// TwinCAT 3 PLC project PLC_wash
// ProgramVersion: 3.1.4022.3
// libraries:
//   Tc2_Standard, * (Beckhoff Automation GmbH)
//   Tc2_System, * (Beckhoff Automation GmbH)
//   Tc3_Module, * (Beckhoff Automation GmbH)
//   VisuSymbols,3.5.10.0,System
// project tree:
//   / GlobalTextList.TcGTLO, PlcTask.TcTTO (not stored), Visualization Manager.TcVMO (not stored)
//   GVLs/ GVL_IO.TcGVL
//   POUs/ MAIN.TcPOU
//   VISUs/ Visualization.TcVIS
// real-time tasks:
//   TASK PlcTask: cycle T#10ms, priority 20, ADS port 350

// ---- GVLs/GVL_IO.TcGVL
{attribute 'qualified_only'}
VAR_GLOBAL
	Fill_valve :BOOL;   // Fill water 
	Drain_valve:BOOL;   // Drain
	SpinMotor  :BOOL;   // Spin Motor
	AgitateMotor: BOOL; // Washing
	PumpOutMotor: BOOL; // Pump motor
    HeaterControl: BOOL; // Optional	
	StartWashing : BOOL;
END_VAR

// ---- POUs/MAIN.TcPOU
PROGRAM MAIN
VAR
	state_Fill:BOOL;
	State_Wash:BOOL;
	State_Rinse:BOOL;
	State_Spin:BOOL;
	Warmwash:BOOL;
	timertime:TIME := T#2000MS;
	Processtime:TON;
	start:BOOL;
	trigger:R_TRIG;
	
	step: INT;
END_VAR

// Your program  comes here ..... 
Processtime(IN:=start, PT:=timertime);
trigger(clk:=gvl_io.StartWashing);


//case: start true dan states true, dan
CASE step OF
	0:
	IF trigger.Q THEN
		start:=TRUE;
		state_Fill:=TRUE;
		gvl_IO.Fill_valve:=TRUE;	
	END_IF
	IF Processtime.Q THEN
		start:=FALSE;
		state_Fill:=FALSE;
		gvl_io.Fill_valve:= FALSE;
		step:=step+1;
	END_IF
	
	1:	
	IF Warmwash THEN
		timertime:=T#6000MS;
		start:=TRUE;
		State_Wash:=TRUE;
		gvl_io.AgitateMotor:=TRUE;
		gvl_io.HeaterControl:=TRUE;
	
	IF	Processtime.Q THEN
		start:=FALSE;
		gvl_io.AgitateMotor:=FALSE;
		gvl_io.HeaterControl:=FALSE;
		step:=step+1;
	END_IF	
		
	END_IF
	
	IF WarmWash=FALSE THEN
		start:=TRUE;
	State_Wash:=TRUE;
	gvl_io.AgitateMotor:=TRUE;
	
	IF	Processtime.Q THEN
		start:=FALSE;
		gvl_io.AgitateMotor:=FALSE;
		step:=step+1;
	END_IF		
	END_IF

	2:
	timertime:=T#2000ms;
	start:=TRUE;
	gvl_io.Drain_valve:=TRUE;
	gvl_io.PumpOutMotor:=TRUE;
	
		IF	Processtime.Q THEN
		start:=FALSE;
		State_Wash:=FALSE;
		gvl_io.Drain_valve:=FALSE;
		gvl_io.PumpOutMotor:=FALSE;
		step:=step+1;
	END_IF	
	
	3:
	start:=TRUE;
	State_Rinse:=TRUE;
	gvl_io.Fill_valve:=TRUE;
	
		IF	Processtime.Q THEN
		start:=FALSE;
		gvl_io.Fill_valve:=FALSE;
		step:=step+1;
	END_IF	
	
	4:
	start:=TRUE;
	gvl_io.AgitateMotor:=TRUE;
	
		IF	Processtime.Q THEN
		start:=FALSE;
		gvl_io.AgitateMotor:=FALSE;
		state_Rinse:=FALSE;
		step:=step+1;
	END_IF	
	5:
	start:=TRUE;
	State_Spin:=TRUE;
	gvl_io.Drain_valve := TRUE;
	gvl_io.SpinMotor:=TRUE;
	gvl_io.PumpOutMotor:=TRUE;
	
		IF	Processtime.Q THEN
		start:=FALSE;
		State_Spin:=FALSE;
		gvl_io.Drain_valve:=FALSE;
		gvl_io.SpinMotor:=FALSE;
		gvl_io.PumpOutMotor:=FALSE;
		step:=0;
	END_IF	
	
END_CASE

END_PROGRAM

// ---- GlobalTextList.TcGTLO
TEXTLIST GlobalTextList
  869 = '%s'
  746 = 'Agitate Motor'
  130 = 'Drain  Valve'
  802 = 'Fill'
  4 = 'Fill Valve'
  757 = 'Heater'
  21 = 'P'
  599 = 'Processtime.ET'
  355 = 'Pump Out Motor'
  679 = 'Rinse'
  546 = 'Spin'
  353 = 'Spin Motor'
  372 = 'Start/Stop'
  733 = 'Warm Washing'
  363 = 'Wash'
END_TEXTLIST

// ---- VISUs/Visualization.TcVIS
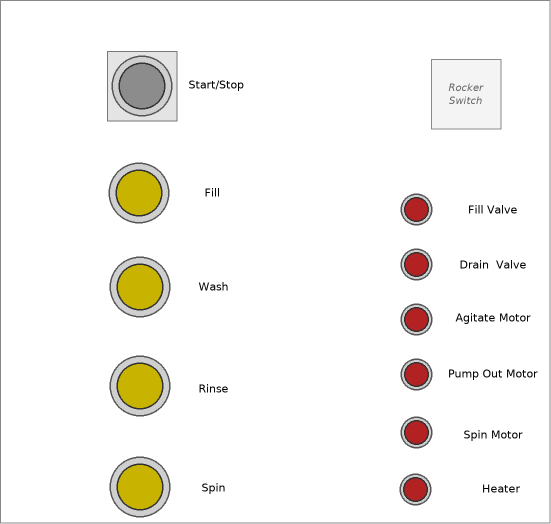
VISUALIZATION Visualization  // 551x524
    Lamp1 (104,158 70x70), variable: MAIN.state_Fill, style: Lamp-Lamp1-Yellow
    Lamp1 (105,252 70x70), variable: MAIN.State_Wash, style: Lamp-Lamp1-Yellow
    Lamp1 (105,351 70x70), variable: MAIN.State_Rinse, style: Lamp-Lamp1-Yellow
    Lamp1 (105,452 70x70), variable: MAIN.State_Spin, style: Lamp-Lamp1-Yellow
    PushSwitch (107,51 70x70), variable: GVL_IO.StartWashing, behaviour: TOGGLE, style: Switch-PushSwitch-Gray
    Lamp1 (397,191 39x37), variable: GVL_IO.Fill_valve, style: Lamp-Lamp1-Red
    Lamp1 (397,246 39x37), variable: GVL_IO.Drain_valve, style: Lamp-Lamp1-Red
    Lamp1 (397,301 39x37), variable: GVL_IO.AgitateMotor, style: Lamp-Lamp1-Red
    Lamp1 (397,356 39x37), variable: GVL_IO.PumpOutMotor, style: Lamp-Lamp1-Red
    Lamp1 (397,414 39x37), variable: GVL_IO.SpinMotor, style: Lamp-Lamp1-Red
    Label (185,178 55x30), "Fill"
    Label (186,272 55x30), "Wash"
    Label (186,374 55x30), "Rinse"
    Label (186,473 55x30), "Spin"
    Label (458,195 70x30), "Fill Valve"
    Label (445,250 96x30), "Drain Valve"
    Label (445,303 96x30), "Agitate Motor"
    Label (445,359 96x30), "Pump Out Motor"
    Label (445,420 96x30), "Spin Motor"
    Label (189,70 55x30), "Start/Stop"
    Lamp1 (396,471 39x37), variable: GVL_IO.HeaterControl, style: Lamp-Lamp1-Red
    Label (453,474 96x30), "Heater"
    RockerSwitch (431,59 70x70), variable: MAIN.Warmwash, behaviour: TOGGLE, style: Switch-RockerSwitch-Gray
END_VISUALIZATION
